// SIMATIC S7-200 SMART project (STEP 7-Micro/WIN SMART), CPU ST30

SYMBOL_TABLE System Symbols
Always_On        SM0.0    // Always ON
Clock_1s         SM0.5    // Clock pulse that is ON for 0.5 s, OFF for 0.5 s, for a duty cycle time of 1 s.
END_SYMBOL_TABLE

ORGANIZATION_BLOCK MAIN:OB1
TITLE=Program Comments
BEGIN
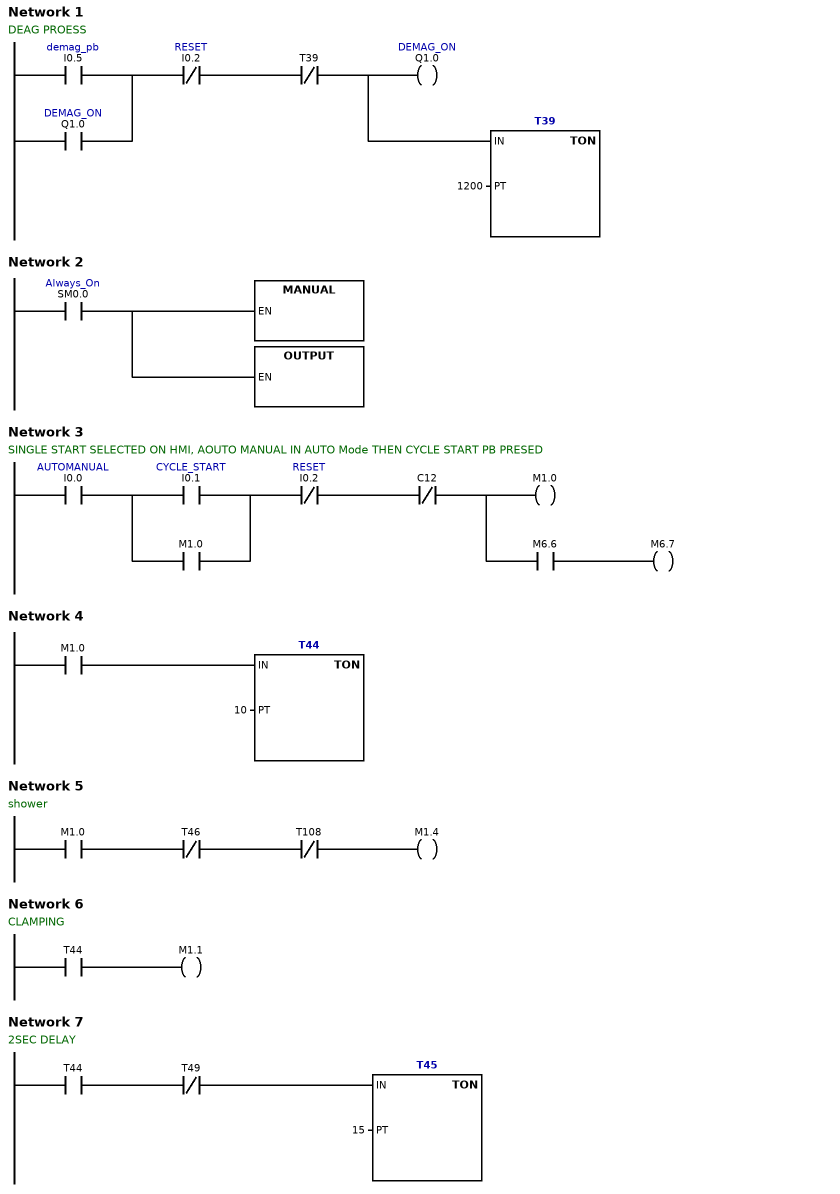
Network 1
// DEAG PROESS
LD     demag_pb:I0.5
O      DEMAG_ON:Q1.0
AN     RESET:I0.2
AN     T39
=      DEMAG_ON:Q1.0
TON    T39, 1200
Network 2
LD     Always_On:SM0.0
CALL   MANUAL:SBR0
CALL   OUTPUT:SBR1
Network 3
// SINGLE START SELECTED ON HMI, AOUTO MANUAL IN AUTO Mode THEN CYCLE START PB PRESED
LD     AUTOMANUAL:I0.0
LD     CYCLE_START:I0.1
O      M1.0
ALD
AN     RESET:I0.2
AN     C12
=      M1.0
A      M6.6
=      M6.7
Network 4
LD     M1.0
TON    T44, 10
Network 5
// shower
LD     M1.0
AN     T46
AN     T108
=      M1.4
Network 6
// CLAMPING 
LD     T44
=      M1.1
Network 7
// 2SEC DELAY
LD     T44
AN     T49
TON    T45, 15
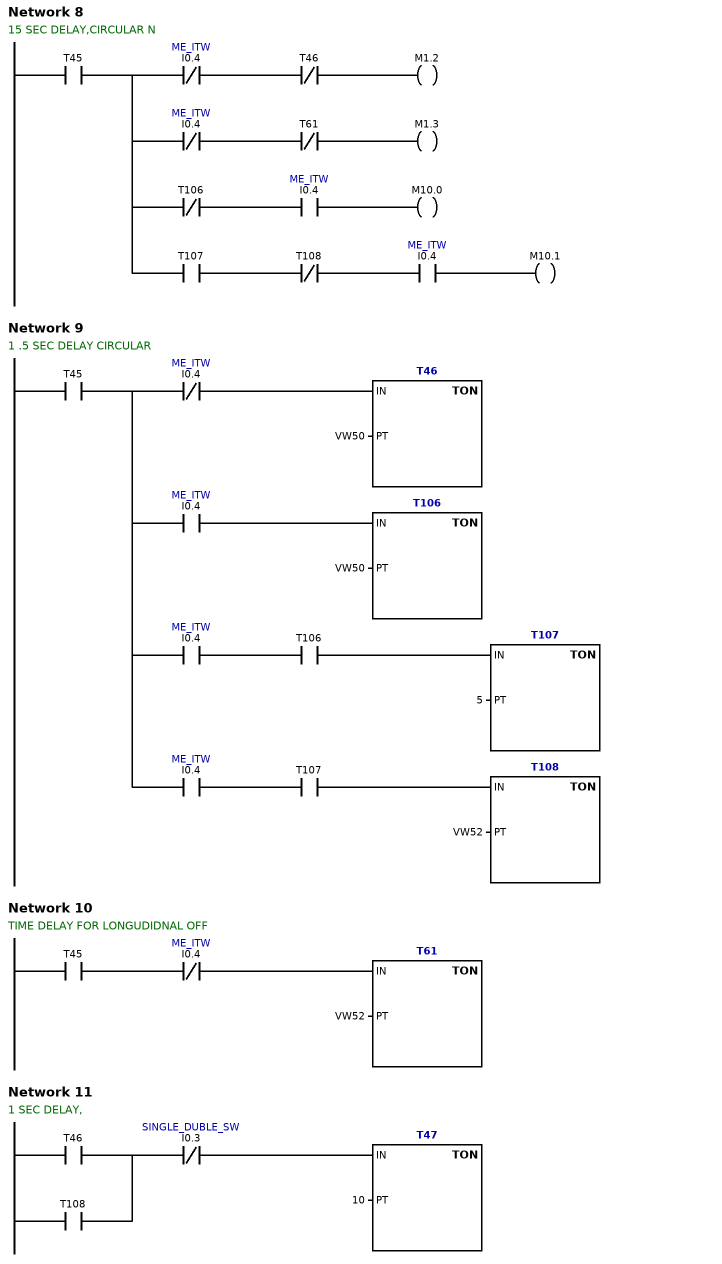
Network 8
// 15 SEC DELAY,CIRCULAR N
LD     T45
LPS
AN     ME_ITW:I0.4
AN     T46
=      M1.2
LRD
AN     ME_ITW:I0.4
AN     T61
=      M1.3
LRD
AN     T106
A      ME_ITW:I0.4
=      M10.0
LPP
A      T107
AN     T108
A      ME_ITW:I0.4
=      M10.1
Network 9
// 1 .5 SEC DELAY CIRCULAR
LD     T45
LPS
AN     ME_ITW:I0.4
TON    T46, VW50
LRD
A      ME_ITW:I0.4
TON    T106, VW50
LRD
A      ME_ITW:I0.4
A      T106
TON    T107, 5
LPP
A      ME_ITW:I0.4
A      T107
TON    T108, VW52
Network 10
// TIME DELAY FOR LONGUDIDNAL OFF
LD     T45
AN     ME_ITW:I0.4
TON    T61, VW52
Network 11
// 1 SEC DELAY,
LD     T46
O      T108
AN     SINGLE_DUBLE_SW:I0.3
TON    T47, 10
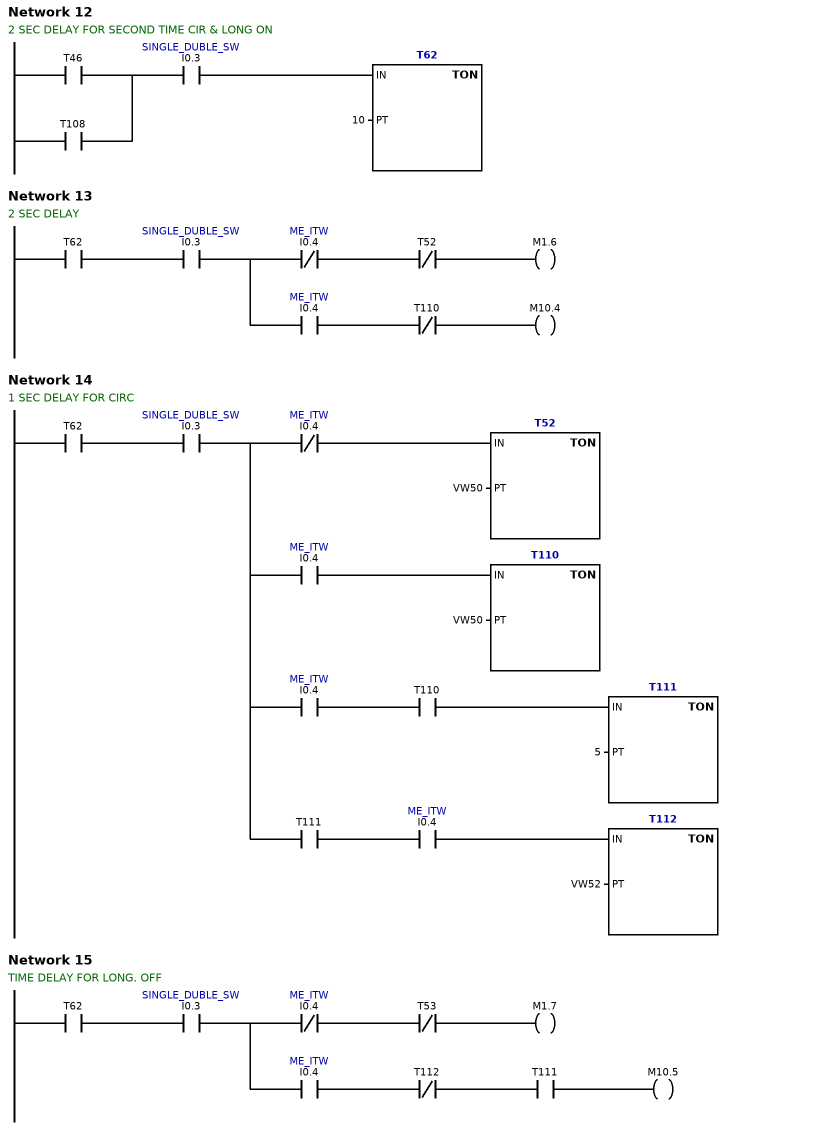
Network 12
// 2 SEC DELAY FOR SECOND TIME CIR & LONG ON
LD     T46
O      T108
A      SINGLE_DUBLE_SW:I0.3
TON    T62, 10
Network 13
// 2 SEC DELAY
LD     T62
A      SINGLE_DUBLE_SW:I0.3
LPS
AN     ME_ITW:I0.4
AN     T52
=      M1.6
LPP
A      ME_ITW:I0.4
AN     T110
=      M10.4
Network 14
// 1 SEC DELAY FOR CIRC
LD     T62
A      SINGLE_DUBLE_SW:I0.3
LPS
AN     ME_ITW:I0.4
TON    T52, VW50
LRD
A      ME_ITW:I0.4
TON    T110, VW50
LRD
A      ME_ITW:I0.4
A      T110
TON    T111, 5
LPP
A      T111
A      ME_ITW:I0.4
TON    T112, VW52
Network 15
// TIME DELAY FOR LONG. OFF
LD     T62
A      SINGLE_DUBLE_SW:I0.3
LPS
AN     ME_ITW:I0.4
AN     T53
=      M1.7
LPP
A      ME_ITW:I0.4
AN     T112
A      T111
=      M10.5
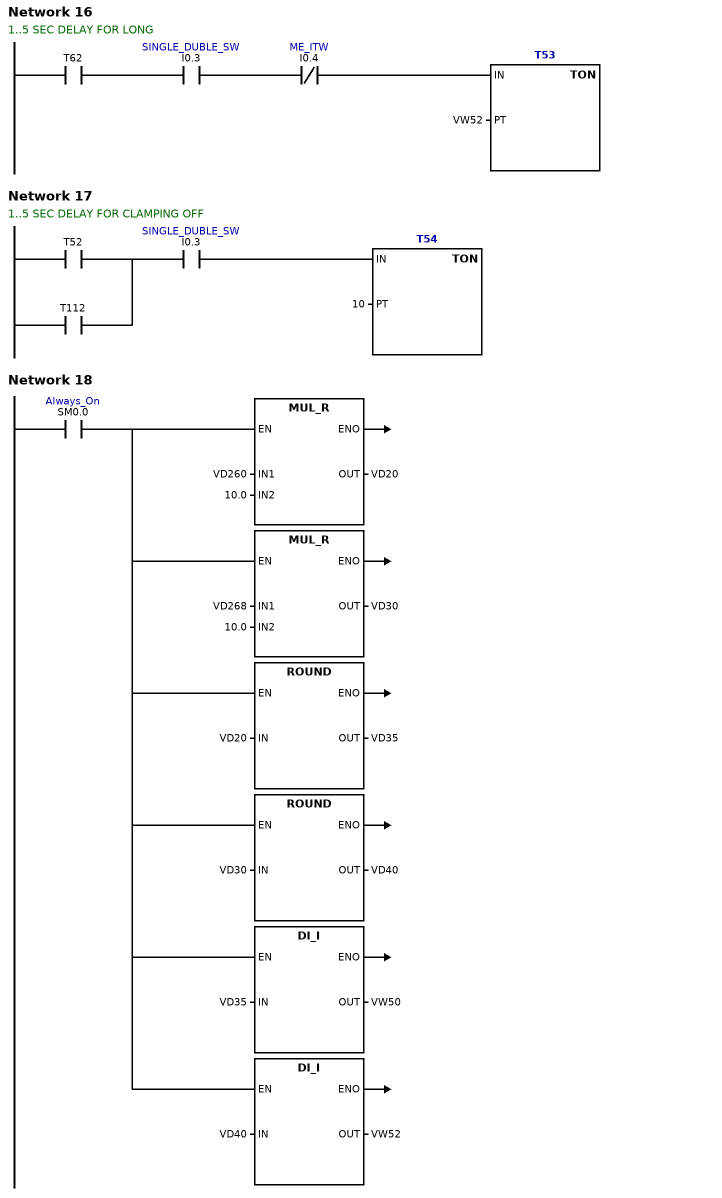
Network 16
// 1..5 SEC DELAY FOR LONG 
LD     T62
A      SINGLE_DUBLE_SW:I0.3
AN     ME_ITW:I0.4
TON    T53, VW52
Network 17
// 1..5 SEC DELAY FOR CLAMPING OFF
LD     T52
O      T112
A      SINGLE_DUBLE_SW:I0.3
TON    T54, 10
Network 18
LD     Always_On:SM0.0
MOVR   VD260, VD20
*R     10.0, VD20
MOVR   VD268, VD30
*R     10.0, VD30
ROUND  VD20, VD35
ROUND  VD30, VD40
DTI    VD35, VW50
DTI    VD40, VW52
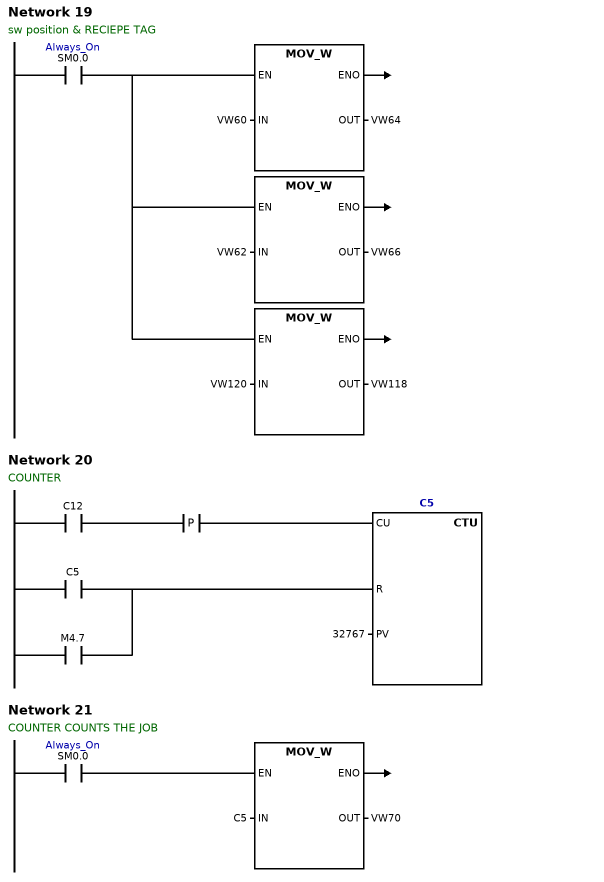
Network 19
// sw position & RECIEPE TAG
LD     Always_On:SM0.0
MOVW   VW60, VW64
MOVW   VW62, VW66
MOVW   VW120, VW118
Network 20
// COUNTER
LD     C12
EU
LD     C5
O      M4.7
CTU    C5, 32767
Network 21
// COUNTER COUNTS THE JOB
LD     Always_On:SM0.0
MOVW   C5, VW70
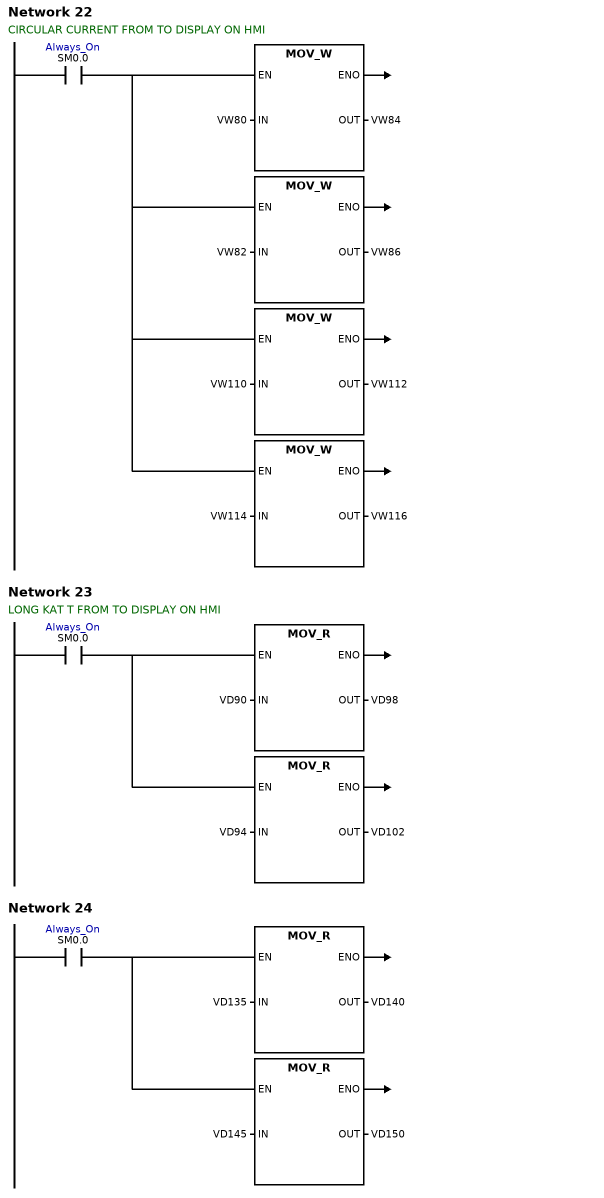
Network 22
// CIRCULAR CURRENT FROM TO DISPLAY ON HMI
LD     Always_On:SM0.0
MOVW   VW80, VW84
MOVW   VW82, VW86
MOVW   VW110, VW112
MOVW   VW114, VW116
Network 23
// LONG KAT T FROM TO DISPLAY ON HMI
LD     Always_On:SM0.0
MOVR   VD90, VD98
MOVR   VD94, VD102
Network 24
LD     Always_On:SM0.0
MOVR   VD135, VD140
MOVR   VD145, VD150
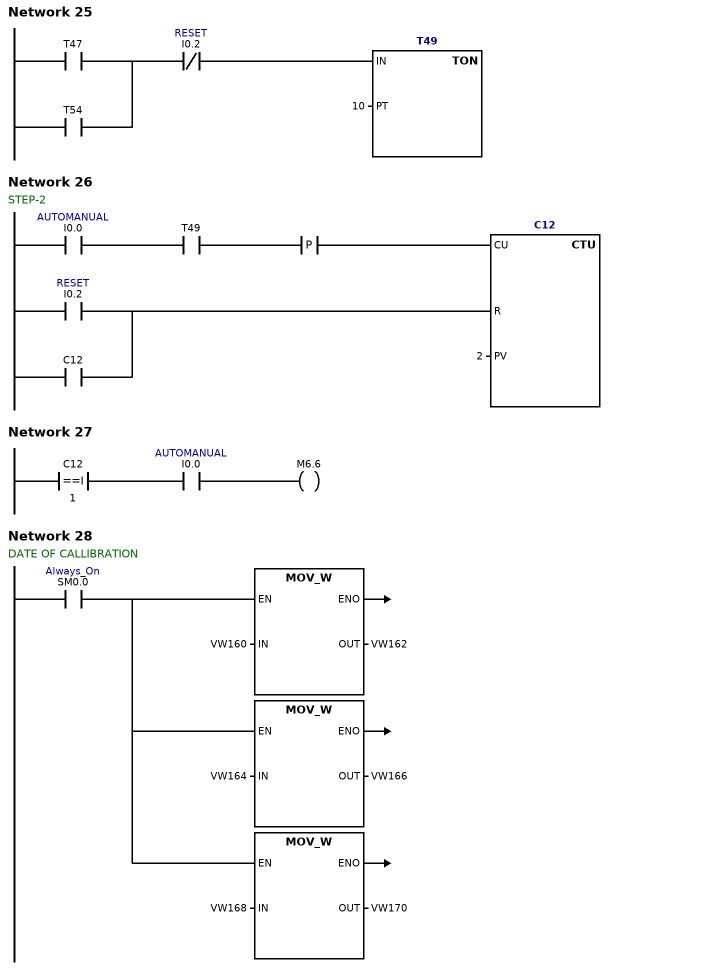
Network 25
LD     T47
O      T54
AN     RESET:I0.2
TON    T49, 10
Network 26
// STEP-2
LD     AUTOMANUAL:I0.0
A      T49
EU
LD     RESET:I0.2
O      C12
CTU    C12, 2
Network 27
LDW=   C12, 1
A      AUTOMANUAL:I0.0
=      M6.6
Network 28
// DATE OF CALLIBRATION
LD     Always_On:SM0.0
MOVW   VW160, VW162
MOVW   VW164, VW166
MOVW   VW168, VW170
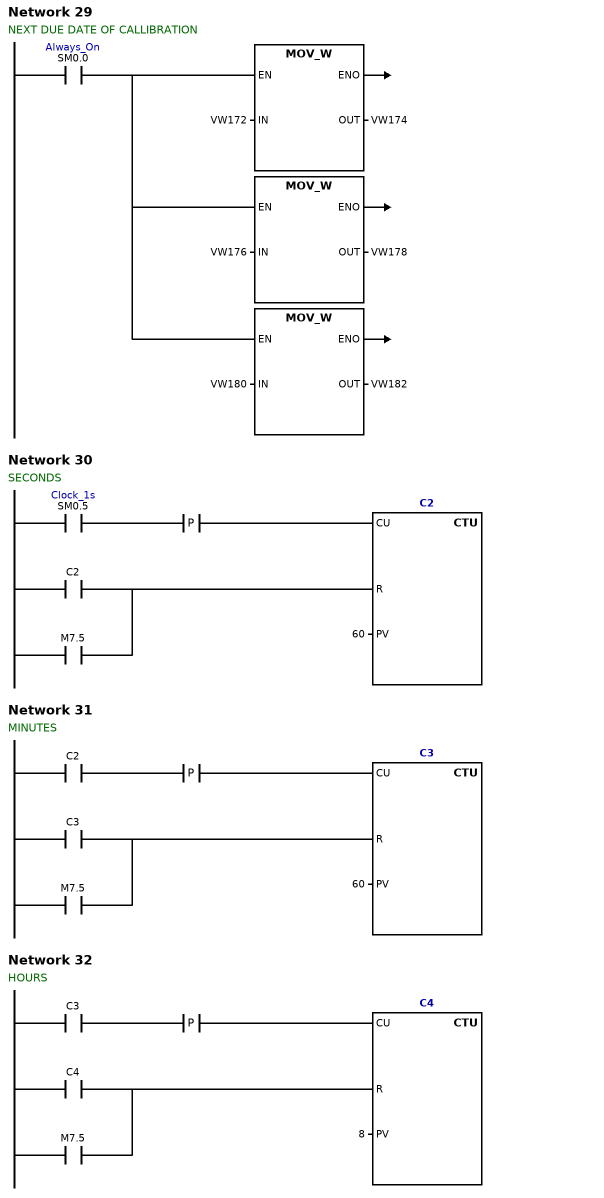
Network 29
// NEXT DUE DATE OF CALLIBRATION
LD     Always_On:SM0.0
MOVW   VW172, VW174
MOVW   VW176, VW178
MOVW   VW180, VW182
Network 30
// SECONDS
LD     Clock_1s:SM0.5
EU
LD     C2
O      M7.5
CTU    C2, 60
Network 31
// MINUTES
LD     C2
EU
LD     C3
O      M7.5
CTU    C3, 60
Network 32
// HOURS
LD     C3
EU
LD     C4
O      M7.5
CTU    C4, 8
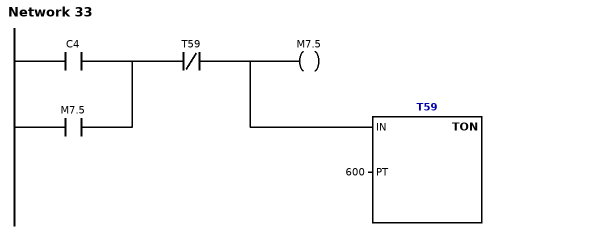
Network 33
LD     C4
O      M7.5
AN     T59
=      M7.5
TON    T59, 600
END_ORGANIZATION_BLOCK

SUBROUTINE_BLOCK MANUAL:SBR0
TITLE=Subroutine Comments
BEGIN
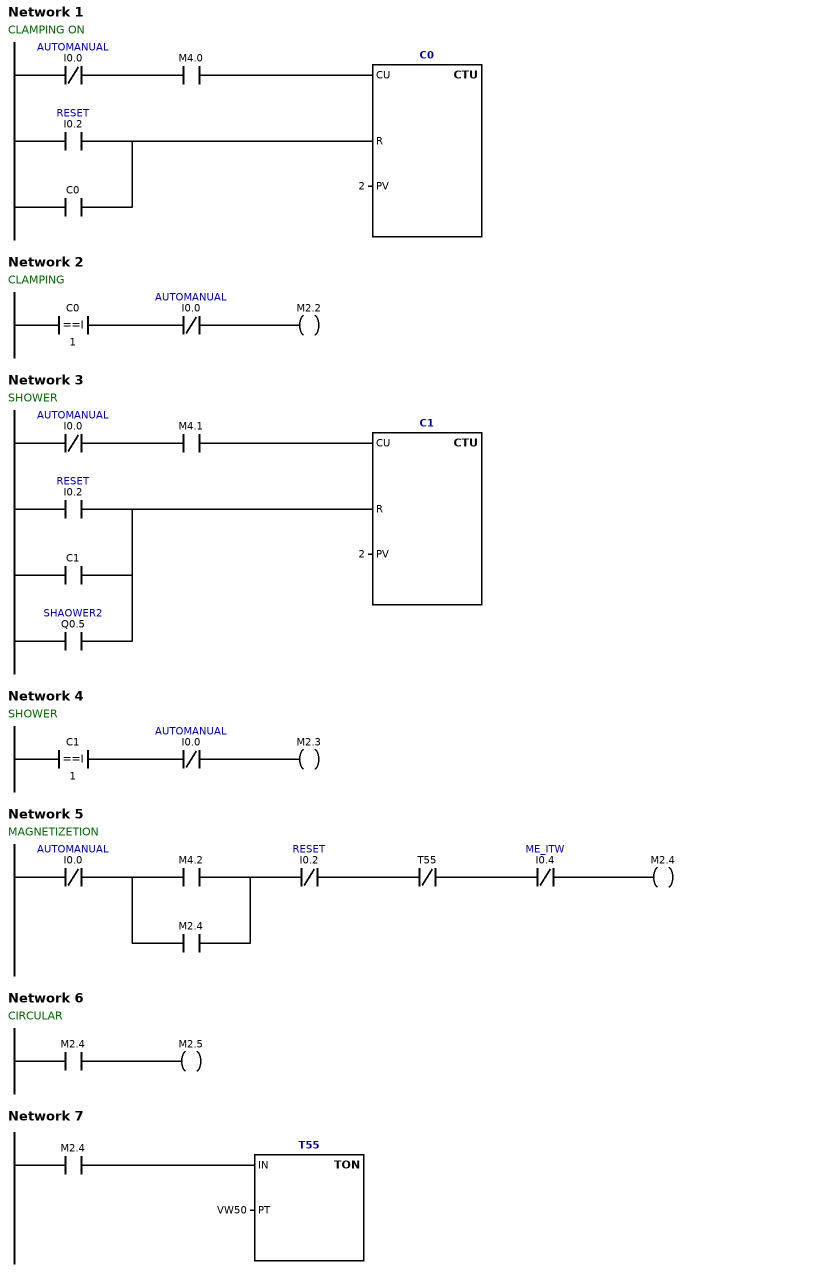
Network 1
// CLAMPING ON
LDN    AUTOMANUAL:I0.0
A      M4.0
LD     RESET:I0.2
O      C0
CTU    C0, 2
Network 2
// CLAMPING
LDW=   C0, 1
AN     AUTOMANUAL:I0.0
=      M2.2
Network 3
// SHOWER
LDN    AUTOMANUAL:I0.0
A      M4.1
LD     RESET:I0.2
O      C1
O      SHAOWER2:Q0.5
CTU    C1, 2
Network 4
// SHOWER
LDW=   C1, 1
AN     AUTOMANUAL:I0.0
=      M2.3
Network 5
// MAGNETIZETION
LDN    AUTOMANUAL:I0.0
LD     M4.2
O      M2.4
ALD
AN     RESET:I0.2
AN     T55
AN     ME_ITW:I0.4
=      M2.4
Network 6
// CIRCULAR
LD     M2.4
=      M2.5
Network 7
LD     M2.4
TON    T55, VW50
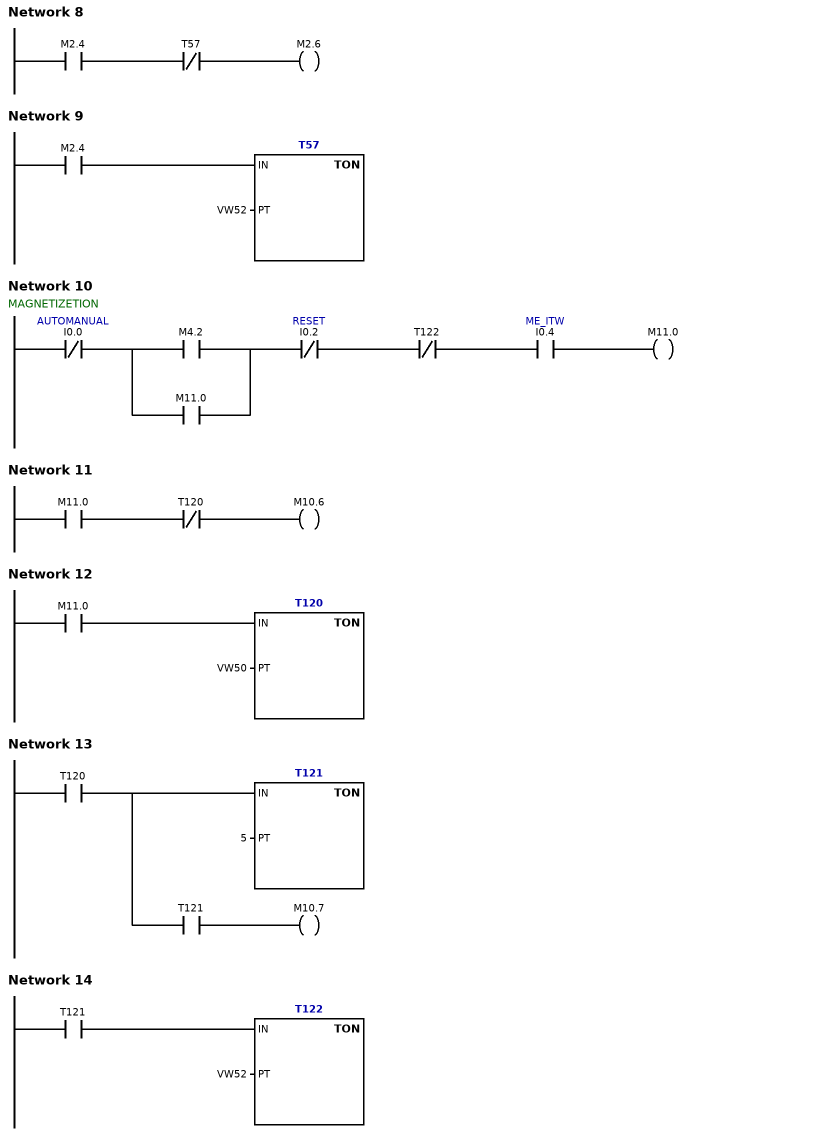
Network 8
LD     M2.4
AN     T57
=      M2.6
Network 9
LD     M2.4
TON    T57, VW52
Network 10
// MAGNETIZETION
LDN    AUTOMANUAL:I0.0
LD     M4.2
O      M11.0
ALD
AN     RESET:I0.2
AN     T122
A      ME_ITW:I0.4
=      M11.0
Network 11
LD     M11.0
AN     T120
=      M10.6
Network 12
LD     M11.0
TON    T120, VW50
Network 13
LD     T120
TON    T121, 5
A      T121
=      M10.7
Network 14
LD     T121
TON    T122, VW52
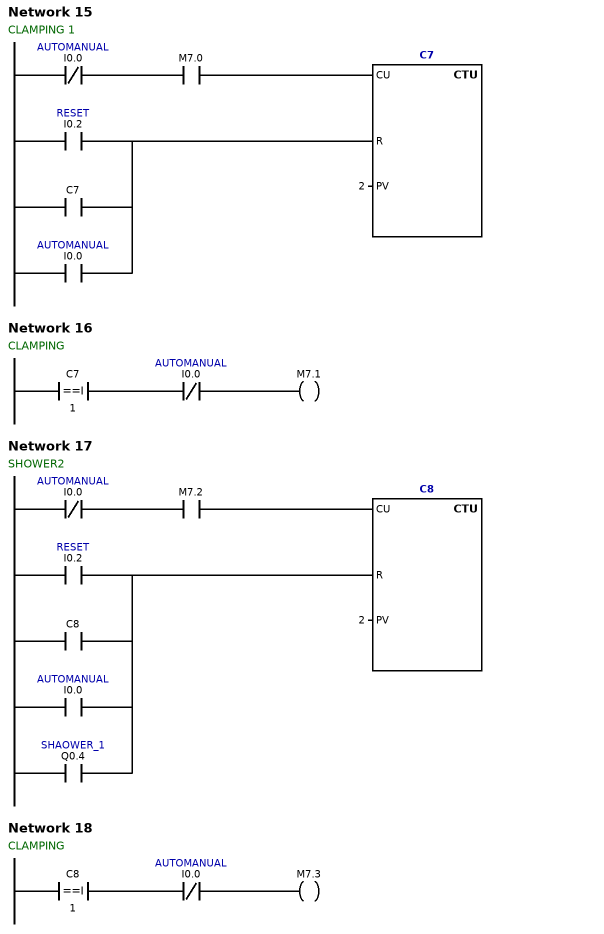
Network 15
// CLAMPING 1
LDN    AUTOMANUAL:I0.0
A      M7.0
LD     RESET:I0.2
O      C7
O      AUTOMANUAL:I0.0
CTU    C7, 2
Network 16
// CLAMPING
LDW=   C7, 1
AN     AUTOMANUAL:I0.0
=      M7.1
Network 17
// SHOWER2
LDN    AUTOMANUAL:I0.0
A      M7.2
LD     RESET:I0.2
O      C8
O      AUTOMANUAL:I0.0
O      SHAOWER_1:Q0.4
CTU    C8, 2
Network 18
// CLAMPING
LDW=   C8, 1
AN     AUTOMANUAL:I0.0
=      M7.3
END_SUBROUTINE_BLOCK

SUBROUTINE_BLOCK OUTPUT:SBR1
TITLE=Subroutine Comments
BEGIN
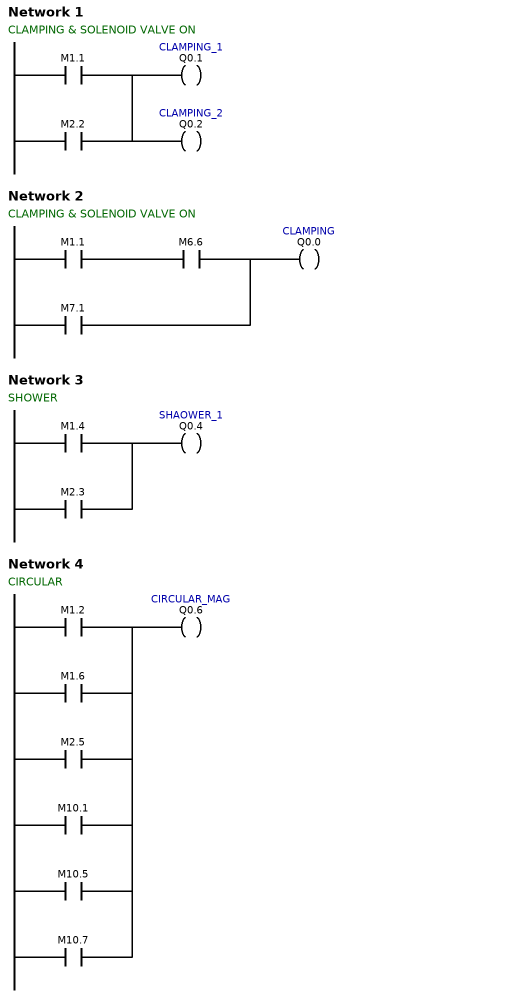
Network 1
// CLAMPING & SOLENOID VALVE ON
LD     M1.1
O      M2.2
=      CLAMPING_1:Q0.1
=      CLAMPING_2:Q0.2
Network 2
// CLAMPING & SOLENOID VALVE ON
LD     M1.1
A      M6.6
O      M7.1
=      CLAMPING:Q0.0
Network 3
// SHOWER
LD     M1.4
O      M2.3
=      SHAOWER_1:Q0.4
Network 4
// CIRCULAR
LD     M1.2
O      M1.6
O      M2.5
O      M10.1
O      M10.5
O      M10.7
=      CIRCULAR_MAG:Q0.6
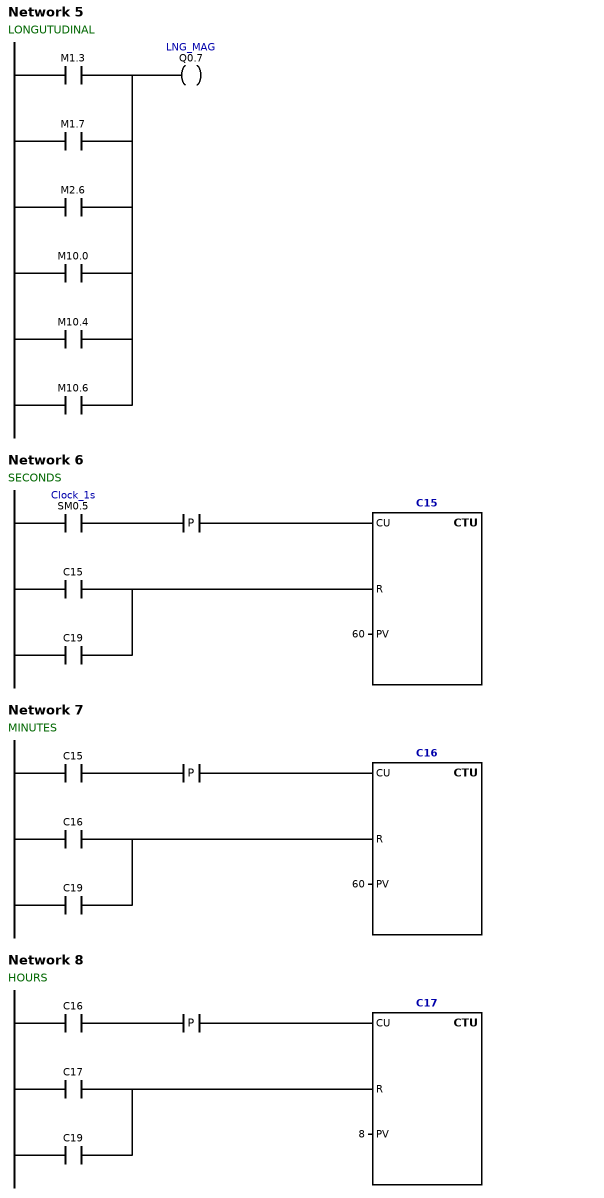
Network 5
// LONGUTUDINAL
LD     M1.3
O      M1.7
O      M2.6
O      M10.0
O      M10.4
O      M10.6
=      LNG_MAG:Q0.7
Network 6
// SECONDS
LD     Clock_1s:SM0.5
EU
LD     C15
O      C19
CTU    C15, 60
Network 7
// MINUTES
LD     C15
EU
LD     C16
O      C19
CTU    C16, 60
Network 8
// HOURS
LD     C16
EU
LD     C17
O      C19
CTU    C17, 8
END_SUBROUTINE_BLOCK
